Fanuc KAREL source: kt00739.KL

PROGRAM KT00739
%STACKSIZE=65535
%PRIORITY=65535
%NOLOCKGROUP
VAR
OUT : INTEGER
-- UNRESOLVED DECLARATIONS (source type spelling not recovered)
-- ARG : ARRAY[4] OF TYPE_0x0018 (type_u16=0x2018)
BEGIN
-- UNSAFE_SOURCE_IR line 7: OUT = native_s16_value(ARG)
END KT00739
